PROGRAM STATION_CYCLE
VAR
END_VAR

grp1();
grp_separate();

ACTION grp_separate:
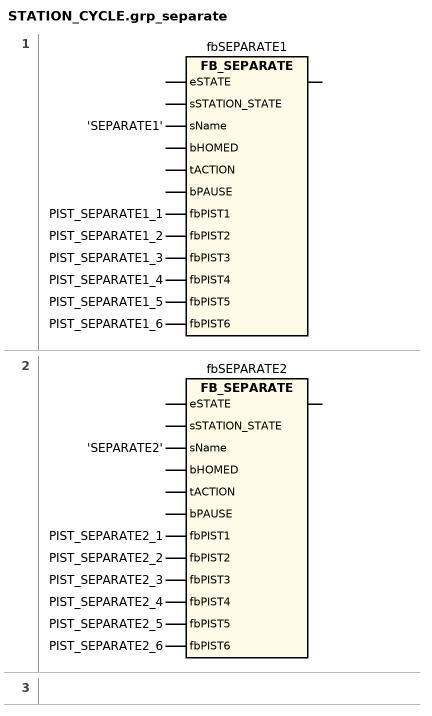
// NETWORK 1
fbSEPARATE1(
    sName := 'SEPARATE1',
    fbPIST1 := PIST_SEPARATE1_1,
    fbPIST2 := PIST_SEPARATE1_2,
    fbPIST3 := PIST_SEPARATE1_3,
    fbPIST4 := PIST_SEPARATE1_4,
    fbPIST5 := PIST_SEPARATE1_5,
    fbPIST6 := PIST_SEPARATE1_6); // FB_SEPARATE

// NETWORK 2
fbSEPARATE2(
    sName := 'SEPARATE2',
    fbPIST1 := PIST_SEPARATE2_1,
    fbPIST2 := PIST_SEPARATE2_2,
    fbPIST3 := PIST_SEPARATE2_3,
    fbPIST4 := PIST_SEPARATE2_4,
    fbPIST5 := PIST_SEPARATE2_5,
    fbPIST6 := PIST_SEPARATE2_6); // FB_SEPARATE

// NETWORK 3
END_ACTION

ACTION grp1:
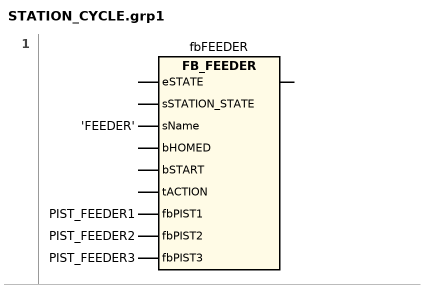
// NETWORK 1
fbFEEDER(sName := 'FEEDER', fbPIST1 := PIST_FEEDER1, fbPIST2 := PIST_FEEDER2, fbPIST3 := PIST_FEEDER3); // FB_FEEDER
END_ACTION

END_PROGRAM

(* stored: Version 1.1.0.1, ProductVersion 3.1.4024.12
   POU STATION_CYCLE: Id {115ce9a0-a0ce-46bf-a813-c5ad1ab48880}, SpecialFunc None
   Action grp_separate: Id {653b6ad7-38a6-4015-9c68-2e96dbef848a}
   Action grp1: Id {b087e6d1-8579-4fe5-b1ea-24bdc6a839eb} *)
